{attribute 'GeneratedUsingTerminal: EK1122-0000-0018'}
{attribute addProperty BoxType "EK1122-0000-0018"}
{attribute addProperty Id "InfoDataAT %I*InfoData_6F19DB2B2"}
{attribute addProperty CRC "532711307"}
{attribute addProperty Size "2"}
TYPE EK1122_1FC0878B EXTENDS EtcSlaveTerminalBase_947E5A46 :
STRUCT
	{attribute addProperty Name "InfoData"}
	InfoData : InfoData_6F19DB2B;
END_STRUCT
END_TYPE

(* stored: Version 1.2.0.0, ProductVersion 3.1.4024.9
   DUT EK1122_1FC0878B: Id {e1baceb9-b604-43d6-84a8-22b6a560e598} *)
